FUNCTION_BLOCK FB_RobotRegionMove_FeedInConveyor EXTENDS FB_ObjectBase_V2 IMPLEMENTS IBasicElement
VAR_INPUT
    Robot     					: REFERENCE TO FB_FanucRobot_Basic_V2;
	LowerConveyor				: REFERENCE TO FB_Motor;
	Input : REFERENCE TO ST_InputTable;

   // Command   : ST_WareHouseWithRobotMove_Command;
    Info	  : ST_RobotRegionMove_Info;
	Stop	  : BOOL;
END_VAR
VAR_OUTPUT
  // Status : ST_WareHouseWithRobotMove_Status;
  
END_VAR
VAR
	_Abort		: BOOL;
	strStatus	: STRING;
	uiResumeStep : UINT;
	
	Area	: E_RobotArea := E_RobotArea.InOutConveyor;
	UseA 	: BOOL;
	UseB	: BOOL;
	
	Get 	:BOOL;
	tonTimeOut	:TON;
	TON_DelayTransMove	:TON;
	_UniqueErrorCode :STRING;
	PreviousStrStatus : STRING;
	PreviousErrorCode : STRING;
END_VAR

SUPER^.A10_StateControl();
A00_BasicUnits();

ACTION A00_BasicUnits:
tonTimeOut(PT:=T#60S);
TON_DelayTransMove(PT :=T#2S);
ErrorID:=2240;
END_ACTION

METHOD M_CheckCommand : BOOL // True : Command is useful
VAR_INPUT
END_VAR
VAR
	
END_VAR
// Check command paremeter is correct
	
	THIS^.Get :=Info.Get;
	UseA := Info.UseA;
	UseB := Info.UseB;

	 //FeedIn/Out conveyor
	 	IF UseA THEN	 
			IF  (Info.A_Position<1 OR  Info.A_Position>3 )THEN
				strStatus:='Wrong command ,Position A Not allow';
				M_CheckCommand:=FALSE;
				RETURN;	
			ELSIF  Info.A_Position=3 AND Get THEN
				strStatus:='Wrong command ,Can Not Get box from FeedOut conveyor ';
				M_CheckCommand:=FALSE;
				RETURN;
			ELSIF 	Info.A_Position <>3 AND NOT Get THEN
				strStatus:='Wrong command ,Can Not Put box to FeedIn conveyor ';
				M_CheckCommand:=FALSE;
				RETURN;				
			END_IF
		END_IF
		
		IF UseB AND ( Info.B_Position<1 OR  Info.B_Position>3 )THEN
			strStatus:='Wrong command ,Position B Not allow';
			M_CheckCommand:=FALSE;
			RETURN;	
		ELSIF UseB AND Info.B_Position=3 AND Get THEN
			strStatus:='Wrong command ,Can Not Get box from FeedOut conveyor ';
			M_CheckCommand:=FALSE;
			RETURN;		
		ELSIF UseB AND Info.B_Position <>3 AND NOT Get THEN
			strStatus:='Wrong command ,Can Not Put box to FeedIn conveyor ';
			M_CheckCommand:=FALSE;
			RETURN;		
		END_IF
		
M_CheckCommand:=TRUE;
END_METHOD

METHOD M_CheckUnitsNotBusy : BOOL
VAR_INPUT
END_VAR
M_CheckUnitsNotBusy := true;
END_METHOD

METHOD M_CheckUnitsReady : BOOL
VAR_INPUT
END_VAR
M_CheckUnitsReady := true;
END_METHOD

METHOD  M_STATE_ABORTED
VAR_INPUT
END_VAR
ERROR :=TRUE;
Busy    := FALSE;
Aborted := TRUE;
Status := strStatus;
UniqueErrorCode:=_UniqueErrorCode;
IF NOT Execute THEN
	eSTATE:=STATE_RESETTING;
END_IF

IF Execute AND Reset THEN
	PreviousStrStatus := strStatus;
	PreviousErrorCode := _UniqueErrorCode;
	uiExecutingStep :=uiResumeStep;
	eSTATE:=STATE_EXECUTING;
END_IF
END_METHOD

METHOD  M_STATE_ABORTING
VAR_INPUT
END_VAR
CASE uiAbortingStep OF
	0 :
		tonTimeOut.IN:=FALSE;
		TON_DelayTransMove.IN :=FALSE;
		LowerConveyor.M_MotorStop();
		IF strStatus = PreviousStrStatus THEN
			_UniqueErrorCode :=PreviousErrorCode;
		END_IF
		uiAbortingStep:=9999;
	
	9999:	_AbortCompleted:=TRUE;
END_CASE

IF _AbortCompleted THEN	
	eSTATE :=STATE_ABORTED;
END_IF
END_METHOD

METHOD  M_STATE_DONE
VAR_INPUT
END_VAR
Busy := FALSE;
Done := TRUE;
IF NOT Execute THEN
    eState := STATE_RESETTING;
END_IF
END_METHOD

METHOD  M_STATE_DORMANT
VAR_INPUT
END_VAR
// Clear FB output
Busy            := FALSE;
Done            := FALSE;
Aborted         := FALSE;
Error           := FALSE;
ErrorID         := 0;
Status          := '';
_ResetCompleted := FALSE;
_Error          := FALSE;
_Executed       := FALSE;

tonTimeOut.IN:=FALSE;
TON_DelayTransMove.IN :=FALSE;
strStatus :='No Error';
uiExecutingStep :=uiResettingStep :=uiResumeStep :=0;
_UniqueErrorCode :='0';
PreviousStrStatus			 :='';
PreviousErrorCode			 :='';

// Wait Execute command
IF Execute THEN
    eState := STATE_EXECUTING;
END_IF
END_METHOD

METHOD  M_STATE_ERROR
VAR_INPUT
END_VAR
ERROR   :=TRUE;
Busy	:=FALSE;
Status := strStatus;
UniqueErrorCode:=_UniqueErrorCode;
IF NOT Execute THEN	
eSTATE:=STATE_RESETTING;
END_IF
END_METHOD

METHOD  M_STATE_EXECUTING
VAR_INPUT
END_VAR
VAR_INST
	BoxReady_1st : BOOL;
	BoxReady_2nd : BOOL;
    uiBothStep : UINT;
    uiSingleClampStep : UINT;	
	Address_A : INT;
	Address_B : INT;
END_VAR
VAR
	WareHouse: INT;
END_VAR
// Set Busy active edit by johnson
Busy := TRUE;
IF THIS^.Stop THEN // Pending the timeout when Stop signal occur
	tonTimeout.IN :=FALSE;
END_IF
// Service Process
CASE uiExecutingStep OF
	0:
        // Clear variable
        uiBothStep := 0;
		uiSingleClampStep :=0;
		BoxReady_1st := 0;
		BoxReady_2nd := 0;
		tonTimeOut.IN:=FALSE;
        // Check command
        IF M_CheckCommand() THEN
            uiExecutingStep := 10;
		ELSE
			_Error:=TRUE;
        END_IF
    10:
        // Start process, check units first
        IF M_CheckUnitsReady() THEN
            uiExecutingStep := 20;
        END_IF
    20:
        // CHeck units not busy state
        IF M_CheckUnitsNotBusy() THEN
            uiExecutingStep := 1000;
        END_IF
   
	1000:   
			// Read   coordinate
			 Area := THIS^.Area;
 			 Address_A := LREAL_TO_INT(Info.A_Position);
			 Address_B := LREAL_TO_INT(Info.B_Position);
			 
			IF UseA AND NOT UseB THEN
				//Only clampA
				uiExecutingStep := 10000;
			ELSIF NOT UseA AND UseB THEN
				//Only ClampB 
				uiExecutingStep := 20000;
			ELSIF UseA AND UseB THEN
				//Both Clamps
				uiExecutingStep := 30000;		
			END_IF
       
    10000: // Only ClampA 
        IF NOT Robot._DI1.Done THEN
            
            
			CASE uiSingleClampStep OF
				
				0://
				
					CASE Address_A OF
						1,2:
							uiSingleClampStep:=1000;
						
						3: 
							uiSingleClampStep:=100;
					END_CASE
				
				100:	
					LowerConveyor.M_MoveBackward();
					IF ( NOT Input.bLowCV_BoxArrived_Sensor) AND ( Input.bLowCV_2ndBoxGap_Sensor) THEN
						tonTimeOut.IN:=FALSE;
						uiSingleClampStep:=200;
					END_IF
					tonTimeOut.IN:=TRUE;
					IF tonTimeOut.Q=TRUE THEN
						strStatus :='Empty Conveyor timeout';
						uiResumeStep:=10000;
						_Abort:=TRUE;
					END_IF
				200:
					TON_DelayTransMove.IN :=TRUE;
					IF TON_DelayTransMove.Q THEN
						LowerConveyor.M_MotorStop();
						uiSingleClampStep:=300;
					END_IF
				
				300:
					TON_DelayTransMove.IN :=FALSE;
					IF 	LowerConveyor.InStopped THEN
						tonTimeOut.IN:=FALSE;
						BoxReady_1st:=TRUE;
						uiSingleClampStep:=9999;
					END_IF
					tonTimeOut.IN:=TRUE;
					IF tonTimeOut.Q=TRUE THEN
						strStatus :='Stop Conveyor timeout';
						_Error:=TRUE;
					END_IF	
				
				1000:
						CASE Address_A OF
							
						1:
							BoxReady_1st:=Input.bUpCV_Block1Detect_Sensor;
						
						2:
							BoxReady_1st:=Input.bUpCV_BoxArrived_Sensor;
						END_CASE						
						
				9999: //
				
			END_CASE
			          		 
				  // Robot Abs move
           		 Robot.M_StartRobotAbsMove(GetBox:=Get,
											UseClampA:=UseA,
											UseClampB:=UseB,
											Area:=Area,
											ClampA_Address:=Address_A,
											ClampB_Address:=Address_B,
											BoxReady_1:=BoxReady_1st,
											BoxReady_2:=BoxReady_2nd);				  
		
        ELSE
			tonTimeOut.IN:=FALSE;
            uiExecutingStep := 10080;
        END_IF
		tonTimeOut.IN:=TRUE;
		IF tonTimeOut.Q=TRUE THEN
			tonTimeOut.IN:=FALSE;
			strStatus :='Reset Robot timeout';
			_Error:=TRUE;
		END_IF	
    10080:
        Robot.M_ResetRobotAbsMove(UseA,UseB); // Clear command and go to place box
		tonTimeOut.IN:=TRUE;
        IF NOT Robot._DI1.Done THEN
			tonTimeOut.IN:=FALSE;
            uiExecutingStep := 80000; 
        END_IF
    	IF tonTimeOut.Q=TRUE THEN
			strStatus :='Reset Robot timeout';
			_Error:=TRUE;
		END_IF	
    
	10090: // Check box 
		
			
   20000: // Only ClampB
        IF NOT Robot._DI1.Done THEN
			
            	CASE uiSingleClampStep OF
				
				0://
				
					CASE Address_B OF
						1,2:
							uiSingleClampStep:=1000;
						
						3: 
							uiSingleClampStep:=100;
					END_CASE
			
				100:	
					LowerConveyor.M_MoveBackward();
					IF (NOT Input.bLowCV_BoxArrived_Sensor) AND  Input.bLowCV_2ndBoxGap_Sensor THEN
						tonTimeOut.IN:=FALSE;
						uiSingleClampStep:=200;
					END_IF
					tonTimeOut.IN:=TRUE;
					IF tonTimeOut.Q=TRUE THEN
						strStatus :='Empty Conveyor timeout';
						uiResumeStep:=20000;
						_Abort:=TRUE;
					END_IF
				200:
					TON_DelayTransMove.IN :=TRUE;
					IF TON_DelayTransMove.Q THEN
						LowerConveyor.M_MotorStop();
						uiSingleClampStep:=300;
					END_IF
				
				300:
					TON_DelayTransMove.IN := FALSE;
					IF 	LowerConveyor.InStopped THEN
						tonTimeOut.IN:=FALSE;
						BoxReady_2nd:=TRUE;
						uiSingleClampStep:=9999;
					END_IF
					tonTimeOut.IN:=TRUE;
					IF tonTimeOut.Q=TRUE THEN
						strStatus :='Stop Conveyor timeout';
						_Error:=TRUE;
					END_IF	
				
				1000:
						CASE Address_B OF
							
						1:
							BoxReady_2nd:=Input.bUpCV_Block1Detect_Sensor;
						
						2:
							BoxReady_2nd:=Input.bUpCV_BoxArrived_Sensor;
						END_CASE						
						
				9999 ://
			END_CASE	
		
			
			          		 
				  // Robot Abs move
           		 Robot.M_StartRobotAbsMove( GetBox:=Get,
											UseClampA:=UseA,
											UseClampB:=UseB,
											Area:=Area,
											ClampA_Address:=Address_A,
											ClampB_Address:=Address_B,
											BoxReady_1:=BoxReady_1st,
											BoxReady_2:=BoxReady_2nd);	
        ELSE
			tonTimeOut.IN:=FALSE;
            uiExecutingStep := 20080;
        END_IF
		tonTimeOut.IN:=TRUE;
		IF tonTimeOut.Q=TRUE THEN
			tonTimeOut.IN:=FALSE;
			strStatus :='Reset Robot timeout';
			_Error:=TRUE;
		END_IF	
    20080:
       Robot.M_ResetRobotAbsMove(UseA,UseB);; // Clear command 

        IF NOT Robot._DI1.Done THEN
            uiExecutingStep := 80000; 
        END_IF
		tonTimeOut.IN:=TRUE;
		IF tonTimeOut.Q=TRUE THEN
			strStatus :='Reset Robot timeout';
			_Error:=TRUE;
		END_IF	
		
	
			
		
    30000: // Both Clamps
        		
		
		  CASE uiBothStep OF
           		0://	
					BoxReady_1st := FALSE;
					BoxReady_2nd := FALSE;
					CASE Address_A OF
						1,2:
							uiBothStep:=1000;
						
						3: 
							uiBothStep:=100;
					END_CASE				
				100:	
					LowerConveyor.M_MoveBackward();
					tonTimeOut.IN:=FALSE;
					IF (NOT Input.bLowCV_BoxArrived_Sensor) AND  Input.bLowCV_2ndBoxGap_Sensor THEN
						uiBothStep:=200;
					END_IF
					tonTimeOut.IN:=TRUE;
					IF tonTimeOut.Q=TRUE THEN
						strStatus :='Empty conveyor timeout';
						uiResumeStep:=30000;
						_Abort:=TRUE;
					END_IF	
				200:
					TON_DelayTransMove.IN := TRUE;
					IF TON_DelayTransMove.Q THEN 
						LowerConveyor.M_MotorStop();
						uiBothStep:=300;
					END_IF
				
				300:
					TON_DelayTransMove.IN :=FALSE;
					IF 	LowerConveyor.InStopped THEN
						tonTimeOut.IN:=FALSE;
						BoxReady_1st:=TRUE;
						uiBothStep:=1000;
					END_IF
					tonTimeOut.IN:=TRUE;
					IF tonTimeOut.Q=TRUE THEN
						strStatus :='Stop conveyor timeout';
						_Error:=TRUE;
					END_IF		
				1000:
				
							CASE Address_A OF							
						1:
							BoxReady_1st:=Input.bUpCV_Block1Detect_Sensor;
						
						2:
							BoxReady_1st:=Input.bUpCV_BoxArrived_Sensor;
						END_CASE
						IF Robot._DI1.Notification THEN
							BoxReady_1st:=TRUE;
							uiBothStep:=2000;
						END_IF
						
						
				2000:
						BoxReady_1st:=TRUE;
						CASE Address_B OF
						1,2:
							uiBothStep:=9000;						
						3: 
							uiBothStep:=3000;
					END_CASE	
				
				3000:	
					LowerConveyor.M_MoveBackward();
					IF (NOT Input.bLowCV_BoxArrived_Sensor) AND Input.bLowCV_2ndBoxGap_Sensor THEN
						tonTimeOut.IN:=FALSE;
						uiBothStep:=3200;
					END_IF
					tonTimeOut.IN:=TRUE;
					IF tonTimeOut.Q=TRUE THEN
						strStatus :='Empty conveyor timeout';
						uiResumeStep:=30000;
						_Abort:=TRUE;
					END_IF	
				3200:
					TON_DelayTransMove.IN := TRUE;
					IF TON_DelayTransMove.Q THEN 
						LowerConveyor.M_MotorStop();
						uiBothStep:=3300;
					END_IF					
				
				3300:
						TON_DelayTransMove.IN :=FALSE;
					IF 	LowerConveyor.InStopped THEN
						tonTimeOut.IN:=FALSE;
						BoxReady_2nd:=TRUE;
						uiBothStep:=9999;
					END_IF
					tonTimeOut.IN:=TRUE;
					IF tonTimeOut.Q=TRUE THEN
						strStatus :='Stop conveyor timeout';
						_Error:=TRUE;
					END_IF		
				9000:
							CASE Address_B OF							
						1:
							BoxReady_2nd:=Input.bUpCV_Block1Detect_Sensor ;
						
						2:
							BoxReady_2nd:=Input.bUpCV_BoxArrived_Sensor;
						END_CASE
				
				9999: //Wait		
        // wait reset
        END_CASE

       	  // Robot Abs move
           		 Robot.M_StartRobotAbsMove( GetBox:=Get,
											UseClampA:=UseA,
											UseClampB:=UseB,
											Area:=Area,
											ClampA_Address:=Address_A,
											ClampB_Address:=Address_B,
											BoxReady_1:=BoxReady_1st,
											BoxReady_2:=BoxReady_2nd);	
		
		
        IF Robot._DI1.Done THEN
			tonTimeOut.IN:=FALSE;
            uiExecutingStep := 30080;
        END_IF
		tonTimeOut.IN:=TRUE;
		IF tonTimeOut.Q=TRUE THEN
			tonTimeOut.IN:=FALSE;
			strStatus :='Reset Robot timeout';
			_Error:=TRUE;
		END_IF
    30080: // Check robot command is clear
        
        Robot.M_ResetRobotAbsMove(UseA,UseB);

        IF NOT Robot._DI1.Done THEN
			tonTimeOut.IN:=FALSE;
            uiExecutingStep := 80000; // go to place step
        END_IF    
   		tonTimeOut.IN:=TRUE;
		IF tonTimeOut.Q=TRUE THEN
			strStatus :='Stop Robot timeout';
			_Error:=TRUE;
		END_IF	
   
		
	80000:
		IF UseA THEN
			CASE Address_A OF
			1:
//				IF Input.bUpCV_BoxArrived_Sensor.P_SignalState THEN
//					strStatus :='Box not taken on F1';
//					_Error:=TRUE;
//				END_IF
				 uiExecutingStep :=99000;
			2:	
//				IF Input.bUpCV_Block1Detect_Sensor.P_SignalState THEN
//					strStatus :='Box not taken on F2';
//					_Error:=TRUE;
//				END_IF	
					uiExecutingStep :=99000;

			3:
				uiExecutingStep :=81000;			
			END_CASE
		END_IF
		IF UseB THEN
			CASE Address_B OF
			1:
//				IF Input.bUpCV_BoxArrived_Sensor.P_SignalState THEN
//					strStatus :='Box not taken on F1';
//					_Error:=TRUE;
//				END_IF
				 uiExecutingStep :=99000;
			2:	
//				IF Input.bUpCV_Block1Detect_Sensor.P_SignalState THEN
//					strStatus :='Box not taken on F2';
//					_Error:=TRUE;
//				END_IF	
					uiExecutingStep :=99000;

			3:
				uiExecutingStep :=81000;			
			END_CASE
		END_IF
		
	81000:
			LowerConveyor.M_MoveBackward();
			tonTimeOut.IN:=FALSE;
			IF (NOT Input.bLowCV_BoxArrived_Sensor) AND ( Input.bLowCV_2ndBoxGap_Sensor) THEN
						uiExecutingStep:=81100;
			END_IF
			tonTimeOut.IN:=TRUE;
			IF tonTimeOut.Q=TRUE THEN
				strStatus :='Empty conveyor timeout';
				_Error:=TRUE;
			END_IF	
	81100:		
//			TON_DelayTransMove.IN := TRUE;
//			IF TON_DelayTransMove.Q THEN
			LowerConveyor.M_MotorStop();
			uiExecutingStep:=81200;
//			END_IF
				
	81200:
			TON_DelayTransMove.IN := false;
			IF 	LowerConveyor.InStopped THEN
				tonTimeOut.IN:=FALSE;
				uiExecutingStep:=99000;
			END_IF
			tonTimeOut.IN:=TRUE;
			IF tonTimeOut.Q=TRUE THEN
				strStatus :='Stop conveyor timeout';
				_Error:=TRUE;
			END_IF		
					
    99000: // process done
          Status    := 'Process completed';
      	  _Executed := TRUE;
END_CASE
IF _Executed THEN
    eState := STATE_DONE;
ELSIF _Error THEN
//	FUN_UniqueErrorCodeGenerator(iErrorID := ErrorID,UinqueErrorCode=>_UniqueErrorCode);
    eState := STATE_ERROR;
ELSIF NOT Execute THEN
    eState := STATE_RESETTING;
END_IF
IF _Abort OR Abort THEN
//	FUN_UniqueErrorCodeGenerator(iErrorID := ErrorID,UinqueErrorCode=>_UniqueErrorCode);
	eSTATE:=STATE_ABORTING;
END_IF
END_METHOD

METHOD  M_STATE_RESETTING
VAR_INPUT
END_VAR
Error :=FALSE;
Done :=FALSE;
Busy := FALSE;


CASE uiResettingStep OF
	
	0:
		tonTimeOut.IN:=FALSE;
		TON_DelayTransMove.IN :=FALSE;
		Robot.M_ResetAllCommand();
		Robot.M_ResetRobotAbsMove(TRUE,TRUE);
		uiResettingStep:=100;
		
	100:
	
		LowerConveyor.M_MotorStop();	
		uiResettingStep:=9999;
	9999:
		_ResetCompleted:=TRUE;
END_CASE
IF _ResetCompleted THEN
	eSTATE:=STATE_DORMANT;
END_IF
END_METHOD

END_FUNCTION_BLOCK

(* stored: Version 1.1.0.1, ProductVersion 3.1.4024.13
   POU FB_RobotRegionMove_FeedInConveyor: Id {cd8bd8a9-d86e-4b34-8910-74681dca6828}, SpecialFunc None
   Folder Method: Id {f940c14f-a193-43ef-a764-d96fd3358e04}
   Folder State: Id {a707b132-c9f0-4a5f-913f-d7b237cbd8f9}
   Action A00_BasicUnits: Id {120d4666-5217-4d96-bc4e-5d19af630e3b}
   Method M_CheckCommand: Id {30c0fce4-a158-4e70-a9aa-05f0490a2517}
   Method M_CheckUnitsNotBusy: Id {0cf24628-5ae2-4bca-9f09-7436e46e9c5d}
   Method M_CheckUnitsReady: Id {05dde86b-f1cc-44fa-8f73-f937439c11e0}
   Method M_STATE_ABORTED: Id {afc65392-e382-4fc3-9f42-baaf8e8a0aaa}
   Method M_STATE_ABORTING: Id {f0cef012-79ee-4067-91f4-a2c95ef7d209}
   Method M_STATE_DONE: Id {0b8f2cfa-be64-4ea1-bdb5-076e32c52515}
   Method M_STATE_DORMANT: Id {193cdfcc-ab79-435d-b6e9-23d4cdcc560a}
   Method M_STATE_ERROR: Id {61f673ec-0700-4b92-9961-46f4e9b460de}
   Method M_STATE_EXECUTING: Id {125187c8-53dc-40c0-97b4-fc67e9cc0069}
   Method M_STATE_RESETTING: Id {62c4f63b-f932-4a79-9176-8414b8de07ae} *)
